// TIA Portal project "WASH_TON_Tom" (V19)

(* hardware
DEVICE "SIMATIC 1200 station_1"  S71200.Device
   slot 0: "S7-1200 rack"  Rack  V1.0
   slot 1: "PLC_1"  CPU 1214C DC/DC/DC  6ES7 214-1AG40-0XB0  V4.0
   slot 3: "AQ1 x 12 bits_1"  6ES7 232-4HA30-0XB0  V1.0
*)

// ===== PLC "PLC_1"  CPU 1214C DC/DC/DC =====

VAR_GLOBAL   // PLC tag table "Default tag table"
   "PUSHBUTTON" AT %I0.0 : Bool;   // Pushbutton Wash Cycle
   "SWITCH_CLAMP1" AT %I0.1 : Bool;   // Limit Switch Clamp 1
   "SWITCH_CLAMP2" AT %I0.2 : Bool;   // Limit Switch Clamp 2
   "SOLENOID_CLAMP1" AT %Q0.0 : Bool;   // Clamp 1 Solenoid
   "SOLENOID_CLAMP2" AT %Q0.1 : Bool;   // Clamp 2 Solenoid
   "WASH_VALVE" AT %Q0.2 : Bool;   // Spray Wash Valve
END_VAR

// folder: System blocks/Program resources

DATA_BLOCK "WASH_DELAY"   // DB1
{ S7_Optimized_Access := 'TRUE' }
AUTHOR : Simatic
FAMILY : IEC
NAME : IEC_TMR
VERSION : 1.0
// stored: InstanceOfName IEC_TIMER
"IEC_TIMER"
BEGIN
END_DATA_BLOCK

// folder: (top level)

ORGANIZATION_BLOCK "Main"   // OB1, SCL, ProgramCycle
TITLE = "Main Program Sweep (Cycle)"
{ S7_Optimized_Access := 'TRUE' }
VERSION : 0.1
BEGIN

   //START pushbuttons to turn On CLAMP solenoids
   IF "PUSHBUTTON" THEN
       "SOLENOID_CLAMP1":=1;
       "SOLENOID_CLAMP2":=1;
   ELSE
       "SOLENOID_CLAMP1":=0;
       "SOLENOID_CLAMP2" := 0;
   END_IF;


   //Timer structure for time to wash when PUSHBUTTON, CLAMP 1 and CLAMP
   ////2 switches are closed
   "WASH_DELAY".TON(IN := "PUSHBUTTON" & "SWITCH_CLAMP1" & "SWITCH_CLAMP2",
                    PT := T#5000ms);

   //Turn On WASH valve when PUSHBUTTON, CLAMP 1 and CLAMP 2 switches are
   ////closed and timer in not complete
   IF "PUSHBUTTON" & "SWITCH_CLAMP1" & "SWITCH_CLAMP2" & NOT "WASH_DELAY".Q THEN
       "WASH_VALVE" := 1;
   ELSE;
       "WASH_VALVE":= 0;
   END_IF;
END_ORGANIZATION_BLOCK